(* IEC 61131-3 sources: ml2plc/benchmarks/st (part 8) *)

VAR
    (* Merged variables from all regions *)
    buffer_0 : ARRAY[0..63] OF REAL;
    buffer_1 : ARRAY[0..63] OF REAL;
    h_new_0 : ARRAY[0..63] OF REAL;
    h_new_3 : ARRAY[0..63] OF REAL;
    h_state_0 : ARRAY[0..63] OF REAL;
    h_state_3 : ARRAY[0..63] OF REAL;
    r_gate_0 : ARRAY[0..63] OF REAL;
    r_gate_3 : ARRAY[0..63] OF REAL;
    u_gate_0 : ARRAY[0..63] OF REAL;
    u_gate_3 : ARRAY[0..63] OF REAL;

    (* Temporary computation variables *)
    i : DINT;
    j : DINT;
    t : DINT;
    sum : REAL;
    (* Computation helpers *)
    max_val : REAL;
    exp_val : REAL;
    exp_sum : REAL;
    (* Spatial loop variables *)
    oc : DINT;
    oh : DINT;
    ow : DINT;
    ic : DINT;
    kh : DINT;
    kw : DINT;
    ih : DINT;
    iw : DINT;
    (* Transpose loop variables *)
    t2_d0 : DINT;
    t2_d1 : DINT;
    t2_d2 : DINT;
END_VAR

(* Forward pass execution *)

(* Region: r0 [ACYCLIC] *)
(* Acyclic Region r0 *)
(* Layer 0: GRU (hidden_size=64, input_size=1, seq_len=1) *)
(* Generating output: Y, linear_before_reset=1 *)

(* Initialize states to zero *)
FOR j := 0 TO 63 DO
    h_state_0[j] := 0.0;
END_FOR;

(* Process 1 timesteps *)
FOR t := 0 TO 0 DO

    (* Reset Gate *)
    FOR j := 0 TO 63 DO
        sum := 0.0;
        FOR i := 0 TO 0 DO
            sum := sum + input_data * weights_0_r[j * 1 + i] ;
        END_FOR;
        FOR i := 0 TO 63 DO
            sum := sum + h_state_0[i] * recurrent_0_r[j * 64 + i] ;
        END_FOR;
    sum := sum + bias_0_r[j];
    r_gate_0[j] := 1.0 / (1.0 + EXP(-sum));
    END_FOR;

    (* Update Gate *)
    FOR j := 0 TO 63 DO
        sum := 0.0;
        FOR i := 0 TO 0 DO
            sum := sum + input_data * weights_0_u[j * 1 + i] ;
        END_FOR;
        FOR i := 0 TO 63 DO
            sum := sum + h_state_0[i] * recurrent_0_u[j * 64 + i] ;
        END_FOR;
    sum := sum + bias_0_u[j];
    u_gate_0[j] := 1.0 / (1.0 + EXP(-sum));
    END_FOR;

    (* Candidate (lbr=1): h'_t = tanh(Wx + r_t * (Rh + Rb_h) + Wb_h) *)
    FOR j := 0 TO 63 DO
        sum := 0.0;
        FOR i := 0 TO 0 DO
            sum := sum + input_data * weights_0_h[j * 1 + i] ;
        END_FOR;
        exp_val := 0.0;
        FOR i := 0 TO 63 DO
            exp_val := exp_val + h_state_0[i] * recurrent_0_h[j * 64 + i] ;
        END_FOR;
        sum := sum + r_gate_0[j] * (exp_val + bias_r_0_h[j]);
        sum := sum + bias_w_0_h[j];
    exp_val := EXP(2.0 * sum);
    h_new_0[j] := (exp_val - 1.0) / (exp_val + 1.0);
    END_FOR;

    (* Hidden state: h_t = u_t * h_{t-1} + (1 - u_t) * h'_t *)
    FOR j := 0 TO 63 DO
        h_state_0[j] := u_gate_0[j] * h_state_0[j] + (1.0 - u_gate_0[j]) * h_new_0[j];
    END_FOR;

    (* Y output: Full sequence *)
    FOR j := 0 TO 63 DO
        buffer_0[t * 64 + j] := h_state_0[j];
    END_FOR;
END_FOR;

(* Layer 1: Squeeze *)
FOR i := 0 TO 63 DO
    buffer_1[i] := buffer_0[i];
END_FOR;

(* Layer 2: Transpose perm=(1, 0, 2)  (1, 1, 64) -> (1, 1, 64) *)
FOR t2_d0 := 0 TO 0 DO
    FOR t2_d1 := 0 TO 0 DO
        FOR t2_d2 := 0 TO 63 DO
            buffer_0[t2_d0 * 64 + t2_d1 * 64 + t2_d2] := buffer_1[t2_d1 * 64 + t2_d0 * 64 + t2_d2];
        END_FOR;
    END_FOR;
END_FOR;

(* Layer 3: GRU (hidden_size=64, input_size=64, seq_len=1) *)
(* Generating output: Y, linear_before_reset=1 *)

(* Initialize states to zero *)
FOR j := 0 TO 63 DO
    h_state_3[j] := 0.0;
END_FOR;

(* Process 1 timesteps *)
FOR t := 0 TO 0 DO

    (* Reset Gate *)
    FOR j := 0 TO 63 DO
        sum := 0.0;
        FOR i := 0 TO 63 DO
            sum := sum + buffer_0[t * 64 + i] * weights_3_r[j * 64 + i] ;
        END_FOR;
        FOR i := 0 TO 63 DO
            sum := sum + h_state_3[i] * recurrent_3_r[j * 64 + i] ;
        END_FOR;
    sum := sum + bias_3_r[j];
    r_gate_3[j] := 1.0 / (1.0 + EXP(-sum));
    END_FOR;

    (* Update Gate *)
    FOR j := 0 TO 63 DO
        sum := 0.0;
        FOR i := 0 TO 63 DO
            sum := sum + buffer_0[t * 64 + i] * weights_3_u[j * 64 + i] ;
        END_FOR;
        FOR i := 0 TO 63 DO
            sum := sum + h_state_3[i] * recurrent_3_u[j * 64 + i] ;
        END_FOR;
    sum := sum + bias_3_u[j];
    u_gate_3[j] := 1.0 / (1.0 + EXP(-sum));
    END_FOR;

    (* Candidate (lbr=1): h'_t = tanh(Wx + r_t * (Rh + Rb_h) + Wb_h) *)
    FOR j := 0 TO 63 DO
        sum := 0.0;
        FOR i := 0 TO 63 DO
            sum := sum + buffer_0[t * 64 + i] * weights_3_h[j * 64 + i] ;
        END_FOR;
        exp_val := 0.0;
        FOR i := 0 TO 63 DO
            exp_val := exp_val + h_state_3[i] * recurrent_3_h[j * 64 + i] ;
        END_FOR;
        sum := sum + r_gate_3[j] * (exp_val + bias_r_3_h[j]);
        sum := sum + bias_w_3_h[j];
    exp_val := EXP(2.0 * sum);
    h_new_3[j] := (exp_val - 1.0) / (exp_val + 1.0);
    END_FOR;

    (* Hidden state: h_t = u_t * h_{t-1} + (1 - u_t) * h'_t *)
    FOR j := 0 TO 63 DO
        h_state_3[j] := u_gate_3[j] * h_state_3[j] + (1.0 - u_gate_3[j]) * h_new_3[j];
    END_FOR;

    (* Y output: Full sequence *)
    FOR j := 0 TO 63 DO
        buffer_1[t * 64 + j] := h_state_3[j];
    END_FOR;
END_FOR;

(* Layer 4: Squeeze *)
FOR i := 0 TO 63 DO
    buffer_0[i] := buffer_1[i];
END_FOR;

(* Layer 5: Slice starts=[0] ends=[1] axes=[0] steps=[1] *)
FOR i := 0 TO 63 DO
    buffer_1[i] := buffer_0[i];
END_FOR;

(* Layer 6: Squeeze *)
FOR i := 0 TO 63 DO
    buffer_0[i] := buffer_1[i];
END_FOR;

(* Layer 7: Fused Linear + SOFTMAX *)
FOR j := 0 TO 2 DO
    sum := 0.0;
    FOR i := 0 TO 63 DO
        sum := sum + buffer_0[i] * weights_7[i * 3 + j];
    END_FOR;
output_data[j] := sum + bias_7[j];
END_FOR;

(* Softmax: find max *)
max_val := output_data[0];
FOR i := 1 TO 2 DO
    IF output_data[i] > max_val THEN
        max_val := output_data[i];
    END_IF;
END_FOR;

(* Softmax: compute exponentials and sum *)
exp_sum := 0.0;
FOR i := 0 TO 2 DO
    output_data[i] := EXP(output_data[i] - max_val);
    exp_sum := exp_sum + output_data[i];
END_FOR;

(* Softmax: normalize *)
FOR i := 0 TO 2 DO
    output_data[i] := output_data[i] / exp_sum;
END_FOR;

END_FUNCTION_BLOCK

(* ---- LSTM1.st ---- *)
FUNCTION_BLOCK LSTM1_FB

    (* Model Inputs/Outputs *)
VAR_INPUT
    input_data : REAL;
END_VAR

VAR_OUTPUT
    output_data : ARRAY[0..2] OF REAL;
END_VAR

VAR CONSTANT
    weights_0_i : ARRAY[0..13] OF REAL := [1.7646029, 2.10398746, 2.19420409, 2.85117745, 2.16055202, 1.16398978, 2.38905668, 1.93622768, 2.37211347, 2.05923724, 2.07184291, 2.40659809, 1.85348392, 1.46550751];
    recurrent_0_i : ARRAY[0..195] OF REAL := [0.000576734543, -0.064728193, -0.229474142, 0.119997896, -0.164283231, -0.10687881, 0.00255717826, 0.219133809, -0.0489157103, -0.183703557, -0.178844273, -0.103609733, 0.0275776684, -0.0296777617, -0.062614508, -0.0771436915, 0.0896899626, 0.0895774364, 0.189815134, 0.0347544365, -0.0174676906, -0.0817190856, 0.0243962295, 0.334960222, 0.0433544926, -0.182088748, 0.175843984, -0.10707514, -0.150145695, 0.183891252, 0.111980245, 0.0627828985, -0.147839561, -0.0525706112, 0.0347394235, -0.0230819397, 0.0686049238, 0.00395798869, 0.27781266, -0.0588732213, -0.0266887918, -0.127925783, 0.142374918, -0.104131564, -0.160723031, -0.0139416102, -0.168722793, -0.0262295119, 0.17650196, -0.172458112, 0.00135627855, -0.0774556845, 0.159455016, -0.00530624203, -0.0644382387, -0.152365029, -0.0927549601, -0.112561882, -0.292680174, 0.083003141, 0.061565876, -0.193448499, 0.128906399, -0.230080962, -0.146881282, -0.0282424763, -0.0634858757, 0.150845572, 0.137223378, 0.134971917, -0.127772585, 0.134101689, -0.146183997, -0.233403891, -0.12873131, 0.0868265331, 0.0180564541, -0.105182856, 0.028658621, 0.129518211, 0.21366559, -0.0675567836, -0.126807094, 0.161935195, 0.149444073, -0.192710727, 0.0185958147, 0.106863558, -0.025951216, 0.0580620617, -0.165250197, 0.185243592, 0.0948283747, 0.135819331, -0.0535071343, 0.0065646572, 0.0457675159, -0.204936266, -0.0908665061, -0.00491538644, -0.248589352, -0.11005345, -0.17256324, -0.00379209314, 0.206906855, -0.170052305, -0.0253892075, 0.171110764, 0.205887288, 0.0402911864, 0.228318781, -0.15670839, 0.135318071, 0.170188472, 0.0335641392, -0.0742551684, 0.0108798891, -0.00695628999, 0.0800488368, 0.0758683234, -0.0460311845, -0.0776472762, 0.269804597, -0.0211064462, 0.0893205777, 0.149165154, 0.0970312208, 0.065577656, -0.0052809231, 0.0568058826, 0.0516724363, -0.149189889, -0.214029342, -0.172699258, 0.232708037, -0.263906449, -0.100571327, -0.0333746001, 0.0916187018, 0.0182130691, -0.184457019, 0.0465662032, 0.0462989211, -0.114803687, -0.119197458, -0.227103487, -0.104520269, 0.03879641, -0.204443902, -0.0593028851, -0.0257012844, -0.422615975, 0.0192758814, -0.00300307292, -0.10245797, 0.082659021, -0.0408013985, -0.0128996894, 0.203832969, -0.131597847, 0.116076834, 0.179722235, 0.227461934, -0.204238936, 0.00747763738, 0.0572294928, 0.248842061, -0.114522174, -0.0340804122, -0.305497348, -0.0728627667, 0.0237209201, 0.084916085, 0.1503077, 0.0132006183, 0.0112578636, -0.071935989, 0.166337371, 0.313166887, -0.0897402614, -0.121459723, 0.0614761114, -0.00690552918, 0.289917111, 0.0115791969, 0.00816774368, 0.108060516, 0.0134463524, 0.0612930171, 0.0542917848, -0.188401505, -0.0220234953, -0.127558872, -0.0865231603, -0.276588619, 0.0412831046];
    bias_0_i : ARRAY[0..13] OF REAL := [2.74101758, 2.81651473, 2.84015226, 2.87464833, 2.6859808, 2.53950071, 2.30480886, 2.7763083, 2.8194716, 2.57531118, 2.47518826, 2.61789656, 2.86349726, 2.39539218];
    weights_0_f : ARRAY[0..13] OF REAL := [0.0994930863, 0.0641649365, 0.0659053028, 0.310496122, -0.0180274844, 0.322808415, 0.13460508, 0.240409821, -0.116530433, 0.268883735, 0.25171873, -0.09833619, -0.143652007, -0.0315733254];
    recurrent_0_f : ARRAY[0..195] OF REAL := [0.330444783, -0.173340008, 0.254967421, 0.0704038218, -0.0412471928, -0.0736248866, -0.0582156442, 0.264827132, -0.135348827, -0.151846945, 0.147201136, -0.020046128, 0.121957049, 0.0184766762, -0.035969492, 0.214979038, 0.034985669, -0.0914698616, -0.274644732, -0.118142888, -0.072329402, 0.116141282, -0.0775460824, -0.107074298, 0.188645467, 0.0262532309, -0.01786015, -0.177582249, 0.0914361179, -0.0663538873, -0.126395732, 0.190274656, -0.13029708, 0.0349565409, 0.00599929178, -0.0175445545, 0.0534397401, 0.0718531162, -0.0483139753, -0.194458738, -0.177942395, 0.250370353, 0.0809427574, -0.094475016, 0.0201020464, -0.232547686, 0.154627278, -0.126319826, -0.128252268, -0.0414301381, -0.265582263, -0.105202571, 0.0266096219, 0.103950769, 0.00543632219, -0.0411446914, -0.0306149013, 0.118214488, -0.207409427, -0.170016184, -0.103816845, 0.172207311, -0.0409844629, 0.200248569, -0.0824343786, 0.0592869371, -0.104873702, -0.212161154, 0.121348836, -0.246069446, -0.00590592902, -0.0422843099, 0.0221838076, -0.160207316, -0.059986636, -0.0523350127, 0.0444642082, -0.124251254, -0.186150134, 0.189812064, -0.242139742, -0.0229474697, 0.0645030141, -0.330164403, 0.174590722, 0.22291857, -0.0418210812, -0.00272266008, 0.157878622, 0.0499391668, 0.0846408159, 0.044251509, 0.390097201, 0.215889871, -0.0754284114, -0.192033708, 0.00324875629, -0.021857854, -0.0535543226, -0.00242765388, 0.162933871, 0.275477529, -0.167581394, -0.115988724, -0.0286814347, 0.129501134, 0.12484014, 0.208047211, 0.0278468095, -0.00393736223, 0.0883823037, -0.18276149, -0.158388153, 0.048879154, 0.0277039129, -0.226456791, -0.153922215, -0.010512339, -0.00974370819, 0.0585962199, 0.19269748, 0.0625768527, -0.0232846756, 0.115240216, -0.00945046451, -0.0141198356, 0.0863936767, 0.128406003, -0.153853804, -0.0456287339, -0.0161963869, 0.177008197, -0.0338094346, 0.103842638, -0.0772012696, 0.0391664505, -0.102441482, 0.375949144, -0.141388834, -0.102128677, 0.0400450528, 0.0960300937, 0.232614085, -0.22481823, -0.127847955, 0.205337495, 0.0536941029, 0.0942906216, 0.116395243, -0.105362907, 0.0104206018, -0.0666923597, 0.173569486, 0.0731921121, -0.13135536, -0.122527391, 0.0288425498, -0.0800838172, -0.0308797751, -0.0638129413, 0.139135733, 0.221251294, 0.0766317397, 0.0293971449, 0.14400804, 0.020618828, -0.0338013731, 0.005458334, 0.0618240237, 0.069802627, -0.0533334836, 0.148841769, 0.0164494719, 0.145708859, -0.000747919374, -0.118926927, -0.109927036, 0.0274634324, 0.0711366385, -0.13021265, -0.217352301, 0.00355160423, -0.01078388, -0.0556534864, 0.136023626, -0.0307185743, -0.0224579871, 0.171888843, -0.0126242051, -0.267865092, 0.0676492155, -0.0560505316, 0.0436061397, -0.234564736, 0.225381255, -0.052390039];
    bias_0_f : ARRAY[0..13] OF REAL := [1, 1, 1, 1, 1, 1, 1, 1, 1, 1, 1, 1, 1, 1];
    weights_0_g : ARRAY[0..13] OF REAL := [-2.34229517, -2.32814503, 2.32577968, 2.26251554, 2.53180718, 1.75660586, 2.26021814, -2.16270947, 2.35147142, -2.43007803, 2.36410999, -2.14994168, -2.09761143, -2.01521564];
    recurrent_0_g : ARRAY[0..195] OF REAL := [0.197011411, 0.140811816, -0.0704584122, -0.224408999, 0.137365937, 0.0961804166, -0.111454219, -0.0359472893, -0.022525873, 0.150108516, 0.00776077062, -0.0701635852, 0.176175594, 0.0836767107, -0.000441269978, 0.162706494, 0.106402405, -0.085004136, 0.243017554, 0.00783823244, -0.196420699, -0.083119221, -0.124454804, -0.0223690849, 0.147707954, -0.0232024975, -0.0441181734, -0.180246502, 0.127271578, 0.0406352356, -0.310184777, -0.0475495085, -0.114168115, -0.0428367183, -0.0422130637, 0.079991132, -0.0948269218, 0.0646525174, 0.151246294, -0.103934556, 0.270481259, 0.0656000897, 0.118079223, 0.209415779, 0.133592054, 0.0443808399, 0.0772913322, 0.277249038, 0.0463525578, -0.168144971, -0.0694826543, -0.0643159598, -0.157264978, 0.0391626731, 0.0264581516, -0.108926147, -0.28564626, 0.0459530205, -0.0218303576, 0.0933430791, 0.0466043502, -0.133756444, 0.048233483, 0.237016737, -0.0262554046, 0.103112124, -0.14360559, -0.0900861174, 0.0985185802, 0.071286127, 0.0866236538, -0.0114489216, 0.0081570372, 0.241550177, -0.113400564, 0.133206651, -0.238634139, -0.120776102, -0.167593971, 0.0674803853, -0.0602275692, 0.0545502678, 0.264214724, 0.0109876785, 0.0824740976, -0.10173519, 0.149255529, -0.0476797447, -0.0438373312, -0.00293017644, 0.177088961, -0.000368840992, -0.0678661764, 0.0248987675, -0.0175857693, 0.0496837161, 0.113237604, 0.0555472001, 0.176424384, 0.0344088636, 0.098974973, 0.0175531227, 0.0618211925, -0.101261556, 0.253718436, 0.245636374, -0.0530016199, 0.251755565, 0.148425162, 0.172887549, -0.00381163089, 0.15694797, -0.00747951539, 0.148076668, 0.0365314707, 0.0355117097, 0.0647161603, -0.100727312, 0.0157361105, 0.0346665457, -0.000271452853, 0.183791742, -0.108315654, -0.198134542, -0.0578069314, 0.190779716, -0.0121636875, -0.29961288, -0.0891132504, -0.232519448, 0.257404298, 0.0520187765, -0.0969726443, 0.0086794775, 0.13444981, -0.211438641, 0.10638807, -0.131581292, -0.1238693, -0.0368137509, -0.0810189918, 0.0520514995, -0.207933113, 0.0324901342, 0.166393846, 0.0761424527, -0.455920309, 0.186049312, 0.0740808025, -0.0189122111, 0.121391751, 0.0442642644, 0.0528342426, 0.131705567, 0.0730170608, -0.0979448706, 0.207684785, 0.0787197277, 0.0203978382, -0.0731295422, -0.104456186, -0.124274328, -0.0791395754, -0.000315232202, 0.250097781, -0.133824691, -0.114593022, -0.178068653, -0.275633335, -0.0667053908, -0.0451372042, 0.175194591, 0.275403082, -0.0339491852, -0.0600487292, -0.00283062458, 0.0322757736, 0.107725516, 0.0587153733, -0.0354104862, 0.181192473, 0.0315516368, -0.175384775, -0.0669292957, -0.0205022879, -0.0642898977, 0.0416383594, -0.0924772099, -0.0504843593, -0.0402859412, 0.11951346, 0.0680008531, -0.12605074, 0.0118287895, -0.326909035, -0.32161516];
    bias_0_g : ARRAY[0..13] OF REAL := [0.86740756, 0.80473727, -0.533454359, -0.506007135, -0.753907442, -0.628560007, -0.303595394, 0.67129302, -0.678550243, 0.456801444, -0.573267162, 0.39612937, 0.505655825, 0.874825358];
    weights_0_o : ARRAY[0..13] OF REAL := [2.12132359, 2.2544601, 2.55398536, 2.77644467, 2.09850049, 0.887302399, 2.29433942, 2.49491572, 2.11278725, 2.29993463, 1.69805646, 2.34314632, 2.07859206, 1.32838297];
    recurrent_0_o : ARRAY[0..195] OF REAL := [0.201155618, 0.122829393, 0.040503554, -0.0926628262, 0.124385737, -0.22958982, 0.172347263, -0.221145272, 0.0853516608, 0.0291274413, -0.0280814096, -0.190518588, 0.0528567098, 0.0744829997, 0.0556683466, -0.204385594, -0.103495255, 0.0840495229, -0.131675407, 0.275533646, -0.0634665042, 0.0115432534, 0.0413113609, -0.000460955314, -0.0644759983, -0.131666869, -0.0403582007, 0.0563414879, -0.198657185, 0.137730286, 0.0631010458, 0.128757313, -0.0108773336, 0.179526761, 0.0743752867, 0.10352996, -0.0463930517, -0.25410533, 0.140421584, -0.101699516, -0.0459680185, -0.0516057499, 0.0551108867, 0.165605903, 0.0683906227, 0.205677763, -0.283685416, -0.0784754977, -0.250414968, -0.111349992, 0.142669171, 0.0748661608, -0.00997680984, 0.0162650291, -0.0284395609, 0.0322339647, 0.205132037, 0.0982485563, -0.233087271, 0.195560187, 0.246935457, 0.172250465, 0.238188282, 0.20523119, -0.069093965, -0.015963994, 0.0525967851, -0.145711347, -0.0440835319, -0.321948528, 0.134902492, -0.162776783, -0.0756857395, -0.248262838, -0.140946269, -0.0665220022, -0.165792972, 0.0559955202, 0.232785866, 0.153235167, 0.0154741332, -0.106321163, -0.15862225, -0.0243484899, 0.119539082, 0.0498817265, -0.105598211, 0.199151829, -0.0106865596, -0.139399111, 0.123677619, -0.0229433421, 0.13605763, -0.186254904, 0.138141006, -0.148037896, -0.172440469, -0.00630055042, 0.0672231913, 0.0394959562, -0.0886815935, -0.0367173627, 0.0342844129, -0.207525522, 0.00729737058, -0.0447931029, -0.0502327681, 0.0189397596, -0.128502443, -0.0456068814, -0.0894328505, 0.134506643, -0.128105134, -0.0428178012, 0.073702313, 0.106830128, -0.0990154967, 0.173071399, 0.0931131616, -0.0460038558, -0.160104424, 0.0857125297, -0.00716175325, -0.018463688, -0.11364869, 0.121156983, 0.138003901, 0.0736444071, -0.0298461318, 0.0339972153, 0.0677925795, -0.339807481, -0.185039684, 0.0543213338, -0.269918859, 0.17620635, 0.0816234872, -0.0323845074, -0.0793842152, -0.104265533, -0.101521134, -0.13089329, 0.287614942, -0.0393214002, 0.110758066, -0.0322699286, 0.10825, 0.029104596, 0.034731824, 0.120363958, -0.0383349136, 0.0361310504, -0.0554852411, 0.00733422814, 0.265616775, -0.117810011, -0.0236164294, 1.00508332e-05, -0.0917709321, -0.141790077, 0.0957797393, -0.0236193575, 0.162388682, -0.00804271549, -0.111998647, 0.0492993779, -0.00616419362, -0.1226025, 0.0456223972, 0.17451784, -0.0461457893, 0.0314298458, 0.0594536625, -0.00577969383, -0.16125837, -0.0659697652, 0.147188932, 0.185183361, 0.221946463, 0.288733035, -0.0874498338, 0.0054717781, -0.104208693, 0.0302618351, -0.115398958, 0.197354183, 0.0545744747, -0.10205555, 0.0588726699, -0.19939287, 0.115329586, -0.0975958481, 0.162130207, 0.112682283, 0.0758139268, -0.148784816];
    bias_0_o : ARRAY[0..13] OF REAL := [2.77339315, 2.83482409, 2.854352, 2.88252306, 2.68838787, 2.52888417, 2.36249995, 2.80373788, 2.82379198, 2.58746719, 2.46438432, 2.6315937, 2.86537814, 2.41817427];

    weights_4 : ARRAY[0..41] OF REAL := [2.49474716, 1.34455371, -2.6931479, 2.33341742, 0.616050184, -3.20293045, -2.94586587, 1.37416399, 2.88620663, -3.86354971, 1.12581575, 2.85354948, -2.75487614, -0.164035901, 2.7680254, -2.13802457, -0.0319068506, 3.68422723, -2.99955487, 1.3359257, 1.18840313, 2.80718899, -0.00796660036, -3.57020688, -2.67162585, 0.468113005, 3.45838761, 2.74723005, -1.79164493, -2.33013725, -3.20562625, 0.930453718, 2.79915333, 3.11756968, -1.37530851, -2.17833233, 3.8540616, -1.26436961, -3.67381907, 1.91691983, 1.4641217, -3.16504598];
    bias_4 : ARRAY[0..2] OF REAL := [-0.0235006064, 0.576158226, -0.990131021];

END_VAR

VAR
    (* Merged variables from all regions *)
    buffer_0 : ARRAY[0..13] OF REAL;
    buffer_1 : ARRAY[0..13] OF REAL;
    c_state_0 : ARRAY[0..13] OF REAL;
    f_gate_0 : ARRAY[0..13] OF REAL;
    g_gate_0 : ARRAY[0..13] OF REAL;
    h_state_0 : ARRAY[0..13] OF REAL;
    i_gate_0 : ARRAY[0..13] OF REAL;
    o_gate_0 : ARRAY[0..13] OF REAL;

    (* Temporary computation variables *)
    i : DINT;
    j : DINT;
    t : DINT;
    sum : REAL;
    (* Computation helpers *)
    max_val : REAL;
    exp_val : REAL;
    exp_sum : REAL;
    (* Spatial loop variables *)
    oc : DINT;
    oh : DINT;
    ow : DINT;
    ic : DINT;
    kh : DINT;
    kw : DINT;
    ih : DINT;
    iw : DINT;
END_VAR

(* Forward pass execution *)

(* Region: r0 [ACYCLIC] *)
(* Acyclic Region r0 *)
(* Layer 0: LSTM (hidden_size=14, input_size=1, seq_len=1) *)
(* Generating output: Y *)

(* Initialize states to zero *)
FOR j := 0 TO 13 DO
    h_state_0[j] := 0.0;
    c_state_0[j] := 0.0;
END_FOR;

(* Process 1 timesteps *)
FOR t := 0 TO 0 DO

    (* Input Gate *)
    FOR j := 0 TO 13 DO
        sum := 0.0;
        FOR i := 0 TO 0 DO
            sum := sum + input_data * weights_0_i[j * 1 + i] ;
        END_FOR;
        FOR i := 0 TO 13 DO
            sum := sum + h_state_0[i] * recurrent_0_i[j * 14 + i] ;
        END_FOR;
    sum := sum + bias_0_i[j];
    i_gate_0[j] := 1.0 / (1.0 + EXP(-sum));
    END_FOR;

    (* Forget Gate *)
    FOR j := 0 TO 13 DO
        sum := 0.0;
        FOR i := 0 TO 0 DO
            sum := sum + input_data * weights_0_f[j * 1 + i] ;
        END_FOR;
        FOR i := 0 TO 13 DO
            sum := sum + h_state_0[i] * recurrent_0_f[j * 14 + i] ;
        END_FOR;
    sum := sum + bias_0_f[j];
    f_gate_0[j] := 1.0 / (1.0 + EXP(-sum));
    END_FOR;

    (* Cell Gate *)
    FOR j := 0 TO 13 DO
        sum := 0.0;
        FOR i := 0 TO 0 DO
            sum := sum + input_data * weights_0_g[j * 1 + i] ;
        END_FOR;
        FOR i := 0 TO 13 DO
            sum := sum + h_state_0[i] * recurrent_0_g[j * 14 + i] ;
        END_FOR;
    sum := sum + bias_0_g[j];
    exp_val := EXP(2.0 * sum);
    g_gate_0[j] := (exp_val - 1.0) / (exp_val + 1.0);
    END_FOR;

    (* Output Gate *)
    FOR j := 0 TO 13 DO
        sum := 0.0;
        FOR i := 0 TO 0 DO
            sum := sum + input_data * weights_0_o[j * 1 + i] ;
        END_FOR;
        FOR i := 0 TO 13 DO
            sum := sum + h_state_0[i] * recurrent_0_o[j * 14 + i] ;
        END_FOR;
    sum := sum + bias_0_o[j];
    o_gate_0[j] := 1.0 / (1.0 + EXP(-sum));
    END_FOR;

    (* Cell state: c_t = f_t * c_{t-1} + i_t * g_t *)
    FOR j := 0 TO 13 DO
        c_state_0[j] := f_gate_0[j] * c_state_0[j] + i_gate_0[j] * g_gate_0[j];
    END_FOR;

    (* Hidden state: h_t = o_t * tanh(c_t) *)
    FOR j := 0 TO 13 DO
        exp_val := EXP(2.0 * c_state_0[j]);
        h_state_0[j] := o_gate_0[j] * ((exp_val - 1.0) / (exp_val + 1.0));
    END_FOR;

    (* Y output: Full sequence *)
    FOR j := 0 TO 13 DO
        buffer_0[t * 14 + j] := h_state_0[j];
    END_FOR;
END_FOR;

(* Layer 1: Squeeze *)
FOR i := 0 TO 13 DO
    buffer_1[i] := buffer_0[i];
END_FOR;

(* Layer 2: Slice starts=[0] ends=[1] axes=[0] steps=[1] *)
FOR i := 0 TO 13 DO
    buffer_0[i] := buffer_1[i];
END_FOR;

(* Layer 3: Squeeze *)
FOR i := 0 TO 13 DO
    buffer_1[i] := buffer_0[i];
END_FOR;

(* Layer 4: Fused Linear + SOFTMAX *)
FOR j := 0 TO 2 DO
    sum := 0.0;
    FOR i := 0 TO 13 DO
        sum := sum + buffer_1[i] * weights_4[i * 3 + j];
    END_FOR;
output_data[j] := sum + bias_4[j];
END_FOR;

(* Softmax: find max *)
max_val := output_data[0];
FOR i := 1 TO 2 DO
    IF output_data[i] > max_val THEN
        max_val := output_data[i];
    END_IF;
END_FOR;

(* Softmax: compute exponentials and sum *)
exp_sum := 0.0;
FOR i := 0 TO 2 DO
    output_data[i] := EXP(output_data[i] - max_val);
    exp_sum := exp_sum + output_data[i];
END_FOR;

(* Softmax: normalize *)
FOR i := 0 TO 2 DO
    output_data[i] := output_data[i] / exp_sum;
END_FOR;

END_FUNCTION_BLOCK

(* ---- LSTM1_straton.st ---- *)
FUNCTION_BLOCK LSTM1_FB

    (* Model Inputs/Outputs *)
VAR_INPUT
    input_data : REAL;
END_VAR

VAR_OUTPUT
    output_data : ARRAY[0..2] OF REAL;
END_VAR

VAR
    CONSTANT weights_0_i : ARRAY[0..13] OF REAL := [1.7646029, 2.10398746, 2.19420409, 2.85117745, 2.16055202, 1.16398978, 2.38905668, 1.93622768, 2.37211347, 2.05923724, 2.07184291, 2.40659809, 1.85348392, 1.46550751];
    CONSTANT recurrent_0_i : ARRAY[0..195] OF REAL := [0.000576734543, -0.064728193, -0.229474142, 0.119997896, -0.164283231, -0.10687881, 0.00255717826, 0.219133809, -0.0489157103, -0.183703557, -0.178844273, -0.103609733, 0.0275776684, -0.0296777617, -0.062614508, -0.0771436915, 0.0896899626, 0.0895774364, 0.189815134, 0.0347544365, -0.0174676906, -0.0817190856, 0.0243962295, 0.334960222, 0.0433544926, -0.182088748, 0.175843984, -0.10707514, -0.150145695, 0.183891252, 0.111980245, 0.0627828985, -0.147839561, -0.0525706112, 0.0347394235, -0.0230819397, 0.0686049238, 0.00395798869, 0.27781266, -0.0588732213, -0.0266887918, -0.127925783, 0.142374918, -0.104131564, -0.160723031, -0.0139416102, -0.168722793, -0.0262295119, 0.17650196, -0.172458112, 0.00135627855, -0.0774556845, 0.159455016, -0.00530624203, -0.0644382387, -0.152365029, -0.0927549601, -0.112561882, -0.292680174, 0.083003141, 0.061565876, -0.193448499, 0.128906399, -0.230080962, -0.146881282, -0.0282424763, -0.0634858757, 0.150845572, 0.137223378, 0.134971917, -0.127772585, 0.134101689, -0.146183997, -0.233403891, -0.12873131, 0.0868265331, 0.0180564541, -0.105182856, 0.028658621, 0.129518211, 0.21366559, -0.0675567836, -0.126807094, 0.161935195, 0.149444073, -0.192710727, 0.0185958147, 0.106863558, -0.025951216, 0.0580620617, -0.165250197, 0.185243592, 0.0948283747, 0.135819331, -0.0535071343, 0.0065646572, 0.0457675159, -0.204936266, -0.0908665061, -0.00491538644, -0.248589352, -0.11005345, -0.17256324, -0.00379209314, 0.206906855, -0.170052305, -0.0253892075, 0.171110764, 0.205887288, 0.0402911864, 0.228318781, -0.15670839, 0.135318071, 0.170188472, 0.0335641392, -0.0742551684, 0.0108798891, -0.00695628999, 0.0800488368, 0.0758683234, -0.0460311845, -0.0776472762, 0.269804597, -0.0211064462, 0.0893205777, 0.149165154, 0.0970312208, 0.065577656, -0.0052809231, 0.0568058826, 0.0516724363, -0.149189889, -0.214029342, -0.172699258, 0.232708037, -0.263906449, -0.100571327, -0.0333746001, 0.0916187018, 0.0182130691, -0.184457019, 0.0465662032, 0.0462989211, -0.114803687, -0.119197458, -0.227103487, -0.104520269, 0.03879641, -0.204443902, -0.0593028851, -0.0257012844, -0.422615975, 0.0192758814, -0.00300307292, -0.10245797, 0.082659021, -0.0408013985, -0.0128996894, 0.203832969, -0.131597847, 0.116076834, 0.179722235, 0.227461934, -0.204238936, 0.00747763738, 0.0572294928, 0.248842061, -0.114522174, -0.0340804122, -0.305497348, -0.0728627667, 0.0237209201, 0.084916085, 0.1503077, 0.0132006183, 0.0112578636, -0.071935989, 0.166337371, 0.313166887, -0.0897402614, -0.121459723, 0.0614761114, -0.00690552918, 0.289917111, 0.0115791969, 0.00816774368, 0.108060516, 0.0134463524, 0.0612930171, 0.0542917848, -0.188401505, -0.0220234953, -0.127558872, -0.0865231603, -0.276588619, 0.0412831046];
    CONSTANT bias_0_i : ARRAY[0..13] OF REAL := [2.74101758, 2.81651473, 2.84015226, 2.87464833, 2.6859808, 2.53950071, 2.30480886, 2.7763083, 2.8194716, 2.57531118, 2.47518826, 2.61789656, 2.86349726, 2.39539218];
    CONSTANT weights_0_f : ARRAY[0..13] OF REAL := [0.0994930863, 0.0641649365, 0.0659053028, 0.310496122, -0.0180274844, 0.322808415, 0.13460508, 0.240409821, -0.116530433, 0.268883735, 0.25171873, -0.09833619, -0.143652007, -0.0315733254];
    CONSTANT recurrent_0_f : ARRAY[0..195] OF REAL := [0.330444783, -0.173340008, 0.254967421, 0.0704038218, -0.0412471928, -0.0736248866, -0.0582156442, 0.264827132, -0.135348827, -0.151846945, 0.147201136, -0.020046128, 0.121957049, 0.0184766762, -0.035969492, 0.214979038, 0.034985669, -0.0914698616, -0.274644732, -0.118142888, -0.072329402, 0.116141282, -0.0775460824, -0.107074298, 0.188645467, 0.0262532309, -0.01786015, -0.177582249, 0.0914361179, -0.0663538873, -0.126395732, 0.190274656, -0.13029708, 0.0349565409, 0.00599929178, -0.0175445545, 0.0534397401, 0.0718531162, -0.0483139753, -0.194458738, -0.177942395, 0.250370353, 0.0809427574, -0.094475016, 0.0201020464, -0.232547686, 0.154627278, -0.126319826, -0.128252268, -0.0414301381, -0.265582263, -0.105202571, 0.0266096219, 0.103950769, 0.00543632219, -0.0411446914, -0.0306149013, 0.118214488, -0.207409427, -0.170016184, -0.103816845, 0.172207311, -0.0409844629, 0.200248569, -0.0824343786, 0.0592869371, -0.104873702, -0.212161154, 0.121348836, -0.246069446, -0.00590592902, -0.0422843099, 0.0221838076, -0.160207316, -0.059986636, -0.0523350127, 0.0444642082, -0.124251254, -0.186150134, 0.189812064, -0.242139742, -0.0229474697, 0.0645030141, -0.330164403, 0.174590722, 0.22291857, -0.0418210812, -0.00272266008, 0.157878622, 0.0499391668, 0.0846408159, 0.044251509, 0.390097201, 0.215889871, -0.0754284114, -0.192033708, 0.00324875629, -0.021857854, -0.0535543226, -0.00242765388, 0.162933871, 0.275477529, -0.167581394, -0.115988724, -0.0286814347, 0.129501134, 0.12484014, 0.208047211, 0.0278468095, -0.00393736223, 0.0883823037, -0.18276149, -0.158388153, 0.048879154, 0.0277039129, -0.226456791, -0.153922215, -0.010512339, -0.00974370819, 0.0585962199, 0.19269748, 0.0625768527, -0.0232846756, 0.115240216, -0.00945046451, -0.0141198356, 0.0863936767, 0.128406003, -0.153853804, -0.0456287339, -0.0161963869, 0.177008197, -0.0338094346, 0.103842638, -0.0772012696, 0.0391664505, -0.102441482, 0.375949144, -0.141388834, -0.102128677, 0.0400450528, 0.0960300937, 0.232614085, -0.22481823, -0.127847955, 0.205337495, 0.0536941029, 0.0942906216, 0.116395243, -0.105362907, 0.0104206018, -0.0666923597, 0.173569486, 0.0731921121, -0.13135536, -0.122527391, 0.0288425498, -0.0800838172, -0.0308797751, -0.0638129413, 0.139135733, 0.221251294, 0.0766317397, 0.0293971449, 0.14400804, 0.020618828, -0.0338013731, 0.005458334, 0.0618240237, 0.069802627, -0.0533334836, 0.148841769, 0.0164494719, 0.145708859, -0.000747919374, -0.118926927, -0.109927036, 0.0274634324, 0.0711366385, -0.13021265, -0.217352301, 0.00355160423, -0.01078388, -0.0556534864, 0.136023626, -0.0307185743, -0.0224579871, 0.171888843, -0.0126242051, -0.267865092, 0.0676492155, -0.0560505316, 0.0436061397, -0.234564736, 0.225381255, -0.052390039];
    CONSTANT bias_0_f : ARRAY[0..13] OF REAL := [1, 1, 1, 1, 1, 1, 1, 1, 1, 1, 1, 1, 1, 1];
    CONSTANT weights_0_g : ARRAY[0..13] OF REAL := [-2.34229517, -2.32814503, 2.32577968, 2.26251554, 2.53180718, 1.75660586, 2.26021814, -2.16270947, 2.35147142, -2.43007803, 2.36410999, -2.14994168, -2.09761143, -2.01521564];
    CONSTANT recurrent_0_g : ARRAY[0..195] OF REAL := [0.197011411, 0.140811816, -0.0704584122, -0.224408999, 0.137365937, 0.0961804166, -0.111454219, -0.0359472893, -0.022525873, 0.150108516, 0.00776077062, -0.0701635852, 0.176175594, 0.0836767107, -0.000441269978, 0.162706494, 0.106402405, -0.085004136, 0.243017554, 0.00783823244, -0.196420699, -0.083119221, -0.124454804, -0.0223690849, 0.147707954, -0.0232024975, -0.0441181734, -0.180246502, 0.127271578, 0.0406352356, -0.310184777, -0.0475495085, -0.114168115, -0.0428367183, -0.0422130637, 0.079991132, -0.0948269218, 0.0646525174, 0.151246294, -0.103934556, 0.270481259, 0.0656000897, 0.118079223, 0.209415779, 0.133592054, 0.0443808399, 0.0772913322, 0.277249038, 0.0463525578, -0.168144971, -0.0694826543, -0.0643159598, -0.157264978, 0.0391626731, 0.0264581516, -0.108926147, -0.28564626, 0.0459530205, -0.0218303576, 0.0933430791, 0.0466043502, -0.133756444, 0.048233483, 0.237016737, -0.0262554046, 0.103112124, -0.14360559, -0.0900861174, 0.0985185802, 0.071286127, 0.0866236538, -0.0114489216, 0.0081570372, 0.241550177, -0.113400564, 0.133206651, -0.238634139, -0.120776102, -0.167593971, 0.0674803853, -0.0602275692, 0.0545502678, 0.264214724, 0.0109876785, 0.0824740976, -0.10173519, 0.149255529, -0.0476797447, -0.0438373312, -0.00293017644, 0.177088961, -0.000368840992, -0.0678661764, 0.0248987675, -0.0175857693, 0.0496837161, 0.113237604, 0.0555472001, 0.176424384, 0.0344088636, 0.098974973, 0.0175531227, 0.0618211925, -0.101261556, 0.253718436, 0.245636374, -0.0530016199, 0.251755565, 0.148425162, 0.172887549, -0.00381163089, 0.15694797, -0.00747951539, 0.148076668, 0.0365314707, 0.0355117097, 0.0647161603, -0.100727312, 0.0157361105, 0.0346665457, -0.000271452853, 0.183791742, -0.108315654, -0.198134542, -0.0578069314, 0.190779716, -0.0121636875, -0.29961288, -0.0891132504, -0.232519448, 0.257404298, 0.0520187765, -0.0969726443, 0.0086794775, 0.13444981, -0.211438641, 0.10638807, -0.131581292, -0.1238693, -0.0368137509, -0.0810189918, 0.0520514995, -0.207933113, 0.0324901342, 0.166393846, 0.0761424527, -0.455920309, 0.186049312, 0.0740808025, -0.0189122111, 0.121391751, 0.0442642644, 0.0528342426, 0.131705567, 0.0730170608, -0.0979448706, 0.207684785, 0.0787197277, 0.0203978382, -0.0731295422, -0.104456186, -0.124274328, -0.0791395754, -0.000315232202, 0.250097781, -0.133824691, -0.114593022, -0.178068653, -0.275633335, -0.0667053908, -0.0451372042, 0.175194591, 0.275403082, -0.0339491852, -0.0600487292, -0.00283062458, 0.0322757736, 0.107725516, 0.0587153733, -0.0354104862, 0.181192473, 0.0315516368, -0.175384775, -0.0669292957, -0.0205022879, -0.0642898977, 0.0416383594, -0.0924772099, -0.0504843593, -0.0402859412, 0.11951346, 0.0680008531, -0.12605074, 0.0118287895, -0.326909035, -0.32161516];
    CONSTANT bias_0_g : ARRAY[0..13] OF REAL := [0.86740756, 0.80473727, -0.533454359, -0.506007135, -0.753907442, -0.628560007, -0.303595394, 0.67129302, -0.678550243, 0.456801444, -0.573267162, 0.39612937, 0.505655825, 0.874825358];
    CONSTANT weights_0_o : ARRAY[0..13] OF REAL := [2.12132359, 2.2544601, 2.55398536, 2.77644467, 2.09850049, 0.887302399, 2.29433942, 2.49491572, 2.11278725, 2.29993463, 1.69805646, 2.34314632, 2.07859206, 1.32838297];
    CONSTANT recurrent_0_o : ARRAY[0..195] OF REAL := [0.201155618, 0.122829393, 0.040503554, -0.0926628262, 0.124385737, -0.22958982, 0.172347263, -0.221145272, 0.0853516608, 0.0291274413, -0.0280814096, -0.190518588, 0.0528567098, 0.0744829997, 0.0556683466, -0.204385594, -0.103495255, 0.0840495229, -0.131675407, 0.275533646, -0.0634665042, 0.0115432534, 0.0413113609, -0.000460955314, -0.0644759983, -0.131666869, -0.0403582007, 0.0563414879, -0.198657185, 0.137730286, 0.0631010458, 0.128757313, -0.0108773336, 0.179526761, 0.0743752867, 0.10352996, -0.0463930517, -0.25410533, 0.140421584, -0.101699516, -0.0459680185, -0.0516057499, 0.0551108867, 0.165605903, 0.0683906227, 0.205677763, -0.283685416, -0.0784754977, -0.250414968, -0.111349992, 0.142669171, 0.0748661608, -0.00997680984, 0.0162650291, -0.0284395609, 0.0322339647, 0.205132037, 0.0982485563, -0.233087271, 0.195560187, 0.246935457, 0.172250465, 0.238188282, 0.20523119, -0.069093965, -0.015963994, 0.0525967851, -0.145711347, -0.0440835319, -0.321948528, 0.134902492, -0.162776783, -0.0756857395, -0.248262838, -0.140946269, -0.0665220022, -0.165792972, 0.0559955202, 0.232785866, 0.153235167, 0.0154741332, -0.106321163, -0.15862225, -0.0243484899, 0.119539082, 0.0498817265, -0.105598211, 0.199151829, -0.0106865596, -0.139399111, 0.123677619, -0.0229433421, 0.13605763, -0.186254904, 0.138141006, -0.148037896, -0.172440469, -0.00630055042, 0.0672231913, 0.0394959562, -0.0886815935, -0.0367173627, 0.0342844129, -0.207525522, 0.00729737058, -0.0447931029, -0.0502327681, 0.0189397596, -0.128502443, -0.0456068814, -0.0894328505, 0.134506643, -0.128105134, -0.0428178012, 0.073702313, 0.106830128, -0.0990154967, 0.173071399, 0.0931131616, -0.0460038558, -0.160104424, 0.0857125297, -0.00716175325, -0.018463688, -0.11364869, 0.121156983, 0.138003901, 0.0736444071, -0.0298461318, 0.0339972153, 0.0677925795, -0.339807481, -0.185039684, 0.0543213338, -0.269918859, 0.17620635, 0.0816234872, -0.0323845074, -0.0793842152, -0.104265533, -0.101521134, -0.13089329, 0.287614942, -0.0393214002, 0.110758066, -0.0322699286, 0.10825, 0.029104596, 0.034731824, 0.120363958, -0.0383349136, 0.0361310504, -0.0554852411, 0.00733422814, 0.265616775, -0.117810011, -0.0236164294, 1.00508332e-05, -0.0917709321, -0.141790077, 0.0957797393, -0.0236193575, 0.162388682, -0.00804271549, -0.111998647, 0.0492993779, -0.00616419362, -0.1226025, 0.0456223972, 0.17451784, -0.0461457893, 0.0314298458, 0.0594536625, -0.00577969383, -0.16125837, -0.0659697652, 0.147188932, 0.185183361, 0.221946463, 0.288733035, -0.0874498338, 0.0054717781, -0.104208693, 0.0302618351, -0.115398958, 0.197354183, 0.0545744747, -0.10205555, 0.0588726699, -0.19939287, 0.115329586, -0.0975958481, 0.162130207, 0.112682283, 0.0758139268, -0.148784816];
    CONSTANT bias_0_o : ARRAY[0..13] OF REAL := [2.77339315, 2.83482409, 2.854352, 2.88252306, 2.68838787, 2.52888417, 2.36249995, 2.80373788, 2.82379198, 2.58746719, 2.46438432, 2.6315937, 2.86537814, 2.41817427];
    CONSTANT weights_4 : ARRAY[0..41] OF REAL := [2.49474716, 1.34455371, -2.6931479, 2.33341742, 0.616050184, -3.20293045, -2.94586587, 1.37416399, 2.88620663, -3.86354971, 1.12581575, 2.85354948, -2.75487614, -0.164035901, 2.7680254, -2.13802457, -0.0319068506, 3.68422723, -2.99955487, 1.3359257, 1.18840313, 2.80718899, -0.00796660036, -3.57020688, -2.67162585, 0.468113005, 3.45838761, 2.74723005, -1.79164493, -2.33013725, -3.20562625, 0.930453718, 2.79915333, 3.11756968, -1.37530851, -2.17833233, 3.8540616, -1.26436961, -3.67381907, 1.91691983, 1.4641217, -3.16504598];
    CONSTANT bias_4 : ARRAY[0..2] OF REAL := [-0.0235006064, 0.576158226, -0.990131021];
END_VAR

VAR
    (* Merged variables from all regions *)
    buffer_0 : ARRAY[0..13] OF REAL;
    buffer_1 : ARRAY[0..13] OF REAL;
    c_state_0 : ARRAY[0..13] OF REAL;
    f_gate_0 : ARRAY[0..13] OF REAL;
    g_gate_0 : ARRAY[0..13] OF REAL;
    h_state_0 : ARRAY[0..13] OF REAL;
    i_gate_0 : ARRAY[0..13] OF REAL;
    o_gate_0 : ARRAY[0..13] OF REAL;

    (* Temporary computation variables *)
    i : DINT;
    j : DINT;
    t : DINT;
    sum : REAL;
    (* Computation helpers *)
    max_val : REAL;
    exp_val : REAL;
    exp_sum : REAL;
    (* Spatial loop variables *)
    oc : DINT;
    oh : DINT;
    ow : DINT;
    ic : DINT;
    kh : DINT;
    kw : DINT;
    ih : DINT;
    iw : DINT;
END_VAR

(* Forward pass execution *)

(* Region: r0 [ACYCLIC] *)
(* Acyclic Region r0 *)
(* Layer 0: LSTM (hidden_size=14, input_size=1, seq_len=1) *)
(* Generating output: Y *)

(* Initialize states to zero *)
FOR j := 0 TO 13 DO
    h_state_0[j] := 0.0;
    c_state_0[j] := 0.0;
END_FOR;

(* Process 1 timesteps *)
FOR t := 0 TO 0 DO

    (* Input Gate *)
    FOR j := 0 TO 13 DO
        sum := 0.0;
        FOR i := 0 TO 0 DO
            sum := sum + input_data * weights_0_i[j * 1 + i] ;
        END_FOR;
        FOR i := 0 TO 13 DO
            sum := sum + h_state_0[i] * recurrent_0_i[j * 14 + i] ;
        END_FOR;
    sum := sum + bias_0_i[j];
    i_gate_0[j] := 1.0 / (1.0 + EXP(-sum));
    END_FOR;

    (* Forget Gate *)
    FOR j := 0 TO 13 DO
        sum := 0.0;
        FOR i := 0 TO 0 DO
            sum := sum + input_data * weights_0_f[j * 1 + i] ;
        END_FOR;
        FOR i := 0 TO 13 DO
            sum := sum + h_state_0[i] * recurrent_0_f[j * 14 + i] ;
        END_FOR;
    sum := sum + bias_0_f[j];
    f_gate_0[j] := 1.0 / (1.0 + EXP(-sum));
    END_FOR;

    (* Cell Gate *)
    FOR j := 0 TO 13 DO
        sum := 0.0;
        FOR i := 0 TO 0 DO
            sum := sum + input_data * weights_0_g[j * 1 + i] ;
        END_FOR;
        FOR i := 0 TO 13 DO
            sum := sum + h_state_0[i] * recurrent_0_g[j * 14 + i] ;
        END_FOR;
    sum := sum + bias_0_g[j];
    exp_val := EXP(2.0 * sum);
    g_gate_0[j] := (exp_val - 1.0) / (exp_val + 1.0);
    END_FOR;

    (* Output Gate *)
    FOR j := 0 TO 13 DO
        sum := 0.0;
        FOR i := 0 TO 0 DO
            sum := sum + input_data * weights_0_o[j * 1 + i] ;
        END_FOR;
        FOR i := 0 TO 13 DO
            sum := sum + h_state_0[i] * recurrent_0_o[j * 14 + i] ;
        END_FOR;
    sum := sum + bias_0_o[j];
    o_gate_0[j] := 1.0 / (1.0 + EXP(-sum));
    END_FOR;

    (* Cell state: c_t = f_t * c_{t-1} + i_t * g_t *)
    FOR j := 0 TO 13 DO
        c_state_0[j] := f_gate_0[j] * c_state_0[j] + i_gate_0[j] * g_gate_0[j];
    END_FOR;

    (* Hidden state: h_t = o_t * tanh(c_t) *)
    FOR j := 0 TO 13 DO
        exp_val := EXP(2.0 * c_state_0[j]);
        h_state_0[j] := o_gate_0[j] * ((exp_val - 1.0) / (exp_val + 1.0));
    END_FOR;

    (* Y output: Full sequence *)
    FOR j := 0 TO 13 DO
        buffer_0[t * 14 + j] := h_state_0[j];
    END_FOR;
END_FOR;

(* Layer 1: Squeeze *)
FOR i := 0 TO 13 DO
    buffer_1[i] := buffer_0[i];
END_FOR;

(* Layer 2: Slice starts=[0] ends=[1] axes=[0] steps=[1] *)
FOR i := 0 TO 13 DO
    buffer_0[i] := buffer_1[i];
END_FOR;

(* Layer 3: Squeeze *)
FOR i := 0 TO 13 DO
    buffer_1[i] := buffer_0[i];
END_FOR;

(* Layer 4: Fused Linear + SOFTMAX *)
FOR j := 0 TO 2 DO
    sum := 0.0;
    FOR i := 0 TO 13 DO
        sum := sum + buffer_1[i] * weights_4[i * 3 + j];
    END_FOR;
output_data[j] := sum + bias_4[j];
END_FOR;

(* Softmax: find max *)
max_val := output_data[0];
FOR i := 1 TO 2 DO
    IF output_data[i] > max_val THEN
        max_val := output_data[i];
    END_IF;
END_FOR;

(* Softmax: compute exponentials and sum *)
exp_sum := 0.0;
FOR i := 0 TO 2 DO
    output_data[i] := EXP(output_data[i] - max_val);
    exp_sum := exp_sum + output_data[i];
END_FOR;

(* Softmax: normalize *)
FOR i := 0 TO 2 DO
    output_data[i] := output_data[i] / exp_sum;
END_FOR;

END_FUNCTION_BLOCK
